	//Make sure string is not empty before using up an array spot.
	IF (StrLenA(pstData:= ADR(sShortString)) > 0) THEN
		TempArray[ArraySize] := sShortString;
		ArraySize := ArraySize + 1;
	END_IF

	//Remove copied components from long string
	StrDeleteA(
		pby:= ADR(StringIn), 
		iLength:= (iSplitLocation + LEN(SPLIT_CHAR)), 
		iPosition:= 1
	);

	//Check to see if more parameters can fit in array. If not exit loop
	IF (ArraySize > GPL_JSON.MAX_LEVELS) THEN
		EXIT;
	END_IF 
END_WHILE

ArraySize:= ArraySize - 1;

FOR i:= 0 TO ArraySize-1 DO
//reverse the order of the array
	VarNameArray[i+1].Name:= TempArray[ArraySize-i];	
END_FOR

SPLIT_VARNAME:= ArraySize;

END_FUNCTION

// Functions/JSONVALUE_TO_STRING
(*
| Author: Tim Van Meppelen, Pro Electric Inc.
| timv@proelectric.com
| Date: May 4, 2021
| convert a JSON value to string
*)
FUNCTION JSONVALUE_TO_STRING : STRING
VAR_INPUT
	In_JSON:		POINTER TO JSONVAR;
END_VAR

CASE In_JSON^.ValueType OF
JSONVALUETYPE.json_null:
	JSONVALUE_TO_STRING:= 'null';
JSONVALUETYPE.json_boolean:
	IF In_JSON^.Boolean THEN
		JSONVALUE_TO_STRING:= 'true';
	ELSE
		JSONVALUE_TO_STRING:= 'false';
	END_IF
JSONVALUETYPE.json_number:
	JSONVALUE_TO_STRING:= REAL_TO_STRING_X(In_JSON^.Number);
JSONVALUETYPE.json_integer:
	JSONVALUE_TO_STRING:= DINT_TO_STRING(In_JSON^.Integer);
JSONVALUETYPE.json_uinteger:
	CASE IN_JSON^.Format OF
	JSONFORMAT.Hex:
		JSONVALUE_TO_STRING:= UDINT_TO_HEXSTR(In_JSON^.UInteger);
	//TO DO:  other formats
	ELSE
		JSONVALUE_TO_STRING:= UDINT_TO_STRING(In_JSON^.UInteger);		
	END_CASE
JSONVALUETYPE.json_string:
	JSONVALUE_TO_STRING:= In_JSON^.CharString;
END_CASE

END_FUNCTION

// Functions/REAL_TO_STRING_X
(*
| Author: Tim Van Meppelen, Pro Electric Inc.
| timv@proelectric.com
| Date: Nov 2, 2018
| Standard REAL_TO_STRING function will always add a decimal place even if the input is a whole number
| this function will drop the ".0" on the string output
*)
FUNCTION REAL_TO_STRING_X : STRING
VAR_INPUT
	In_REAL:		REAL;
END_VAR
VAR
	TempVar:		STRING;
END_VAR

TempVar:= REAL_TO_STRING(In_REAL);
IF (RIGHT(STR:= TempVar, SIZE:= 2) = '.0') THEN
	REAL_TO_STRING_X:= DELETE(STR:= TempVar, LEN:= 2, POS:= LEN(TempVar) - 1);
ELSE
	REAL_TO_STRING_X:= TempVar;
END_IF

END_FUNCTION

// Functions/UDINT_TO_HEXSTR
(*
| Description:
| This function converts a UDINT (Unsigned Double Integer) value
| to its corresponding hexadecimal string representation (uppercase).
| 
| Example inputs/outputs: 255 -> '0xFF', 419 -> '0x1A3', 305419896 -> '0x12345678', 0 -> '0x0'
| 
| Limitations:
| - The returned string contains only valid hexadecimal digits (0-9, A-F), with '0x' prefix.
| - The output is always in uppercase.
| 
| Author: Fabrizio Morlino
| Date: 20/05/2025
*)
FUNCTION UDINT_TO_HEXSTR : STRING
VAR_INPUT
	udIn	: UDINT;
END_VAR
VAR
    i       : INT;
    nibble  : BYTE;
    result  : STRING(12) := '0x';
    hexchar : ARRAY[0..15] OF STRING(1) := ['0', '1', '2', '3', '4', '5', '6', '7', '8', '9','A', 'B', 'C', 'D', 'E', 'F'];
	xNotSkip: BOOL := FALSE;
END_VAR

// The FOR loop iterates through each nibble (4 bits) of the DWORD,
// starting from the most significant (bits 28-31) to the least significant (bits 0-3).
// 4 BYTE => 8 NIBBLE
FOR i := 7 TO 0 BY -1 DO
	nibble := TO_BYTE(SHR(udIn, i * 4) AND 16#F);
	// To write only the necessary digits (without zero-padding on the left)
	xNotSkip := xNotSkip OR nibble > 0 OR i = 0; //<= 1;
	IF xNotSkip THEN
		result := CONCAT(result, hexchar[nibble]);
	END_IF
END_FOR

UDINT_TO_HEXSTR := result;

END_FUNCTION

// Functions/STRING_TO_JSONVALUE
(*
| Author: Tim Van Meppelen, Pro Electric Inc.
| timv@proelectric.com
| Date: May 4, 2021
| Convert a string to a JSON value
*)
FUNCTION STRING_TO_JSONVALUE
VAR_INPUT
	In_String:		STRING(GPL_JSON.MAX_VALUE_SIZE);
	Out_JSON:		POINTER TO JSONVAR;
END_VAR
VAR
	TempBool:		BOOL;
	TempReal:		REAL;
	TempInt:		DINT;
	TempUint:		UDINT;
	Format:			JSONFORMAT;
END_VAR

IF (Out_JSON^.ValueType = JSONVALUETYPE.json_null) THEN
//if the type is not explicitly configured, make a guess at the type
//NOTE: this is used in JSON_TO_STRUCT to determine variable type
	Out_JSON^.ValueType:= VALUETYPE_FROM_STRING(In_String:= In_String, Format=> Format);
	OUT_JSON^.Format:= Format;	//helper var
END_IF

CASE Out_JSON^.ValueType OF
JSONVALUETYPE.json_null:
	Out_JSON^.Null:= 'null';
JSONVALUETYPE.json_boolean:
	StrToUpperA(pString:= ADR(In_String));
	IF (In_String = 'TRUE') THEN
		TempBool:= TRUE;
	ELSE
		TempBool:= FALSE;
	END_IF
	Out_JSON^.Boolean:= TempBool;
JSONVALUETYPE.json_integer:
	TempInt:= STRING_TO_DINT(In_String);
	Out_JSON^.Integer:= TempInt;
JSONVALUETYPE.json_uinteger:
	IF ISHEX(ADR(In_String)) THEN
		TempUInt:= HEXSTR_TO_UDINT(In_String);
	ELSE
		TempUint:= STRING_TO_UDINT(In_String);
	END_IF
	Out_JSON^.UInteger:= TempUInt;
JSONVALUETYPE.json_number:
	TempReal:= STRING_TO_REAL(In_String);
	Out_JSON^.Number:= TempReal;
JSONVALUETYPE.json_string:
	Out_JSON^.CharString:= In_String;
END_CASE

END_FUNCTION

// Functions/VALUETYPE_FROM_STRING
(*
| Author: Tim Van Meppelen, Pro Electric Inc.
| timv@proelectric.com
| Date: May 4, 2021
| take a guess at what kind of value this is based on what the string looks like
*)
FUNCTION VALUETYPE_FROM_STRING : JSONVALUETYPE
VAR_INPUT
	In_String:		STRING(GPL_JSON.MAX_VALUE_SIZE);
END_VAR
VAR_OUTPUT
	Format:			JSONFORMAT;
END_VAR

IF ISINTEGER(ADR(In_String)) THEN
	VALUETYPE_FROM_STRING:= JSONVALUETYPE.json_integer;
ELSIF ISNUMBER(ADR(In_String)) THEN
	VALUETYPE_FROM_STRING:= JSONVALUETYPE.json_number;
//NOTE:  UInteger type disabled because it's not
//necessarily possible to check for signed/unsigned from a string, where 
//the value could change.  Therefore, json_uinteger type must be manually configured
//ELSIF ISUINTEGER(ADR(In_String)) THEN
//	VALUETYPE_FROM_STRING:= JSONVALUETYPE.json_uinteger;	
ELSIF ISHEX(ADR(In_String)) THEN
	VALUETYPE_FROM_STRING:= JSONVALUETYPE.json_uinteger;
	Format:= JSONFORMAT.Hex;
ELSIF ISBOOLEAN(ADR(In_String)) THEN
	VALUETYPE_FROM_STRING:= JSONVALUETYPE.json_boolean;
ELSIF ISNULL(ADR(In_String)) THEN
	VALUETYPE_FROM_STRING:= JSONVALUETYPE.json_null;
ELSE
	VALUETYPE_FROM_STRING:= JSONVALUETYPE.json_string;
END_IF

END_FUNCTION

// Functions/ISINTEGER
(*
| Author: Tim Van Meppelen, Pro Electric Inc.
| timv@proelectric.com
| Date: Mar 2, 2020
| check if a string contains an integer, allows for "-" at the beginning of the string, and no decimals
*)
FUNCTION ISINTEGER : BOOL
VAR_INPUT
	In:				POINTER TO ARRAY[1..255] OF ASCII;
END_VAR
VAR
	i:				UINT;
	founddecimal:	BOOL;
END_VAR

FOR i:= 1 TO 255 DO
	CASE In^[i] OF 	
	ASCII.NULL:
	//end of string
		EXIT;
	ASCII.MINUS:
	//only allow a "-" in the first position	
		IF (i=1) THEN
			ISINTEGER:= TRUE;
		ELSE
			ISINTEGER:= FALSE;
			EXIT;
		END_IF
	ASCII.DOT:
	//no decimal points allowed in integers
		ISINTEGER:= FALSE;
		EXIT;
	ASCII._0..ASCII._9:
		ISINTEGER:= TRUE;
	ELSE
	//all other characters are not part of numbers
		ISINTEGER:= FALSE;
		EXIT;
	END_CASE
END_FOR

END_FUNCTION

// Functions/ISNUMBER
(*
| Author: Tim Van Meppelen, Pro Electric Inc.
| timv@proelectric.com
| Date: Oct 2, 2018
| check if a string contains a valid number, allows for "-" at the beginning of the string, and one "." character
| update June 9, 2025: allow for scientific notation
*)
FUNCTION ISNUMBER : BOOL
VAR_INPUT
	In:				POINTER TO ARRAY[1..255] OF ASCII;
END_VAR
VAR
    i                   : UINT;
    foundDecimal        : BOOL := FALSE;       // true after first '.'
    foundExponent       : BOOL := FALSE;       // true after first 'e' or 'E'
    insideExponent      : BOOL := FALSE;       // parsing the exponent section
    expSignAllowed      : BOOL := FALSE;       // '+' or '-' allowed only once just after 'e'
    expDigitFound       : BOOL := FALSE;       // at least one digit required after e/E
END_VAR

// -----------------------------------------------------------------------------
// Scan the string until the terminating ASCII.NULL (0x00) or buffer end.
// -----------------------------------------------------------------------------
FOR i := 1 TO 255 DO
    CASE In^[i] OF
    ASCII.NULL :             // reached end of string
        // valid only if we are not still waiting for exponent digits
        ISNUMBER := NOT insideExponent OR expDigitFound;
        RETURN;

    // -------------------------------------------------------------------------
    // Optional leading sign (only '-' is used in literal syntax, '+' is legal
    // in expressions but not required for a constant; keep '-' behaviour).
    // Inside exponent one optional '+' or '-' may follow immediately after 'e'.
    // -------------------------------------------------------------------------
    ASCII.MINUS, ASCII.PLUS :
        IF (i = 1) AND (In^[i] = ASCII.MINUS) THEN
            // leading '-' of mantissa
            ISNUMBER := TRUE;

        ELSIF insideExponent AND expSignAllowed THEN
            // sign belonging to exponent
            expSignAllowed := FALSE;  // consume it
        ELSE
            ISNUMBER := FALSE;
            RETURN;
        END_IF;

    // -------------------------------------------------------------------------
    // Decimal point allowed exactly once and only before the exponent.
    // -------------------------------------------------------------------------
    ASCII.DOT :
        IF foundDecimal OR insideExponent THEN
            ISNUMBER := FALSE; RETURN;
        END_IF;
        foundDecimal := TRUE;

    // -------------------------------------------------------------------------
    // Exponent marker ('e' or 'E') allowed once and must follow at least
    // one digit of the mantissa.
    // -------------------------------------------------------------------------
    ASCII._e_, ASCII._E :
        IF foundExponent THEN
            ISNUMBER := FALSE; RETURN;    // second exponent → invalid
        END_IF;
        foundExponent  := TRUE;
        insideExponent := TRUE;
        expSignAllowed := TRUE;           // allow one optional sign next
        expDigitFound  := FALSE;          // reset digit flag for exponent

    // -------------------------------------------------------------------------
    // Digits are always allowed; in exponent they satisfy the “at least one
    // digit” rule.
    // -------------------------------------------------------------------------
    ASCII._0..ASCII._9 :
        IF insideExponent THEN
            expDigitFound := TRUE;
            expSignAllowed := FALSE;      // any further '+'/'-' now illegal
        END_IF;
        ISNUMBER := TRUE;

    // -------------------------------------------------------------------------
    ELSE        // any other character invalidates the literal
        ISNUMBER := FALSE;
        RETURN;
    END_CASE
END_FOR
// If the loop ends without meeting ASCII.NULL, treat as “not a number”
ISNUMBER := FALSE;

END_FUNCTION

// Functions/ISHEX
(*
| Description:
| This function checks whether the input string is a valid hexadecimal value.
| The string may optionally start with '0x' or '0X'.
| Only characters 0-9, A-F, and a-f are considered valid (after the optional prefix).
| 
| Example inputs: 'FF' -> TRUE, '0xFF' -> TRUE, '1A3' -> TRUE, '0x123G' -> FALSE, '' -> FALSE
| 
| Limitations:
| - The maximum allowed length of the hexadecimal string (excluding '0x') is 8 characters.
| - Returns FALSE if the string is empty or contains invalid characters.
| 
| Author: Fabrizio Morlino
| Date: 20/05/2025
*)
FUNCTION ISHEX : BOOL
VAR_INPUT
	In	: POINTER TO ARRAY[1..255] OF ASCII;
END_VAR
VAR
	i	: UINT;
END_VAR

FOR i:= 1 TO 256 DO
	CASE In^[i] OF
	ASCII.NULL:
	//end of string
		EXIT;
	ASCII._x_:
	//only allow a "x" in the second position	
		IF (i=2) THEN
			ISHEX:= TRUE;
		ELSE
			ISHEX:= FALSE;
			EXIT;
		END_IF		
	ASCII._a_..ASCII._f_:
		ISHEX:= TRUE;
	ASCII._A..ASCII._F:
		ISHEX:= TRUE;
	ASCII._0..ASCII._9:
		ISHEX:= TRUE;
	ELSE // all other characters are not part of numbers
		ISHEX:= FALSE;
		EXIT;		
	END_CASE
END_FOR

END_FUNCTION

// Functions/ISBOOLEAN
(*
| Author: Tim Van Meppelen, Pro Electric Inc.
| timv@proelectric.com
| Date: Oct 2, 2018
| check if a string would convert to a valid boolean variable
*)
FUNCTION ISBOOLEAN : BOOL
VAR_INPUT
	In:			POINTER TO STRING(5);
END_VAR
VAR
	TempVar:	STRING(5);
END_VAR

TempVar:= In^;
StrToUpperA(pString:= ADR(TempVar));

ISBOOLEAN:= (TempVar = 'TRUE') OR (TempVar = 'FALSE');

END_FUNCTION

// Functions/ISNULL
(*
| Author: Tim Van Meppelen, Pro Electric Inc.
| timv@proelectric.com
| Date: June 5, 2025
| check if a string reads null
*)
FUNCTION ISNULL : BOOL
VAR_INPUT
	In:			POINTER TO STRING(4);
END_VAR
VAR
	TempVar:	STRING(4);
END_VAR

TempVar:= In^;
StrToUpperA(pString:= ADR(TempVar));

ISNULL:= (TempVar = 'NULL');

END_FUNCTION

// Functions/HEXSTR_TO_UDINT
(*
| Description:
| This function converts a string representing a hexadecimal number
| into a UDINT (Unsigned Double Integer) value.
| The string may optionally start with '0x' or '0X'.
| 
| Example inputs: 'FF' -> 255, '0xFF' -> 255, '1A3' -> 419, '0x12345678' -> 305419896
| 
| Limitations:
| - The maximum length of the hexadecimal string (excluding '0x') is 8 characters,
|   since a UDINT is a 32-bit integer (2^32 - 1), which corresponds to FFFFFFFF in hexadecimal.
| 
| Author: Fabrizio Morlino
| Date: 20/05/2025
*)
FUNCTION HEXSTR_TO_UDINT : UDINT
VAR_INPUT
    sHex 		: STRING; // Hex string to convert 
END_VAR
VAR_OUTPUT
	xError		: BOOL;
END_VAR
VAR
    i        	: INT;          // Index for iteration
    c        	: BYTE;         // Current character
    digit    	: BYTE;         // Numeric value of the hexadecimal character
    result   	: UDINT := 0;   // Final result
    sHexLen  	: INT;          // Length of the string
    startIdx 	: INT := 0;     // Start index after the prefix
END_VAR

// Removes the '0x' or '0X' prefix if present
IF (LEFT(sHex, 2) = '0x') OR (LEFT(sHex, 2) = '0X') THEN
    startIdx := 2;
END_IF;

sHexLen := LEN(sHex);

// If the string is empty after the prefix
IF sHexLen - startIdx <= 0 THEN
	xError := TRUE;
	RETURN;
END_IF

// If the hexadecimal string is too large for a UDINT
IF sHexLen - startIdx > 8 THEN
	xError := TRUE;
	RETURN;
END_IF

// Iterate through each character of the string
FOR i := startIdx TO sHexLen - 1 DO
    c := sHex[i];
    // Convert the character to a numeric value
    IF (c >= ASCII._0) AND (c <= ASCII._9) THEN
        digit := TO_BYTE(c) - ASCII._0;
    ELSIF (c >= ASCII._A) AND (c <= ASCII._F) THEN
        digit := TO_BYTE(c) - ASCII._A + 10;
    ELSIF (c >= ASCII._a_) AND (c <= ASCII._f_) THEN
        digit := TO_BYTE(c) - ASCII._a_ + 10;
    ELSE
        // Invalid character
		xError := TRUE;
        RETURN;
    END_IF;

    // Accumulate the result
    result := result * 16 + TO_UDINT(digit);
END_FOR;

// Returns the converted value
HEXSTR_TO_UDINT := result;

END_FUNCTION

// Functions/DWORD_TO_HEXSTR
(*
| Description:
| This function converts a UDINT (Unsigned Double Integer) value
| to its corresponding hexadecimal string representation (uppercase).
| 
| Example inputs/outputs: 255 -> '0xFF', 419 -> '0x1A3', 305419896 -> '0x12345678', 0 -> '0x0'
| modified to always return 4 decimals for unicode characters
| Limitations:
| - The returned string contains only valid hexadecimal digits (0-9, A-F), with '0x' prefix.
| - The output is always in uppercase.
| 
| Author: Fabrizio Morlino
| Date: 20/05/2025
*)
FUNCTION DWORD_TO_HEXSTR : STRING
VAR_INPUT
	dWIn	: DWORD;
END_VAR
VAR
    i       : INT;
    nibble  : BYTE;
    result  : STRING(12) := '0x';
    hexchar : ARRAY[0..15] OF STRING(1) := ['0', '1', '2', '3', '4', '5', '6', '7', '8', '9','A', 'B', 'C', 'D', 'E', 'F'];
	xNotSkip: BOOL := FALSE;
END_VAR

// The FOR loop iterates through each nibble (4 bits) of the DWORD,
// starting from the most significant (bits 28-31) to the least significant (bits 0-3).
// 4 BYTE => 8 NIBBLE
FOR i := 7 TO 0 BY -1 DO
	nibble := TO_BYTE(SHR(dWIn, i * 4) AND 16#F);
	// To write only the necessary digits (without zero-padding on the left)
	xNotSkip := xNotSkip OR nibble > 0 OR i = 0; //<= 1;
	IF xNotSkip THEN
		result := CONCAT(result, hexchar[nibble]);
	END_IF
END_FOR

DWORD_TO_HEXSTR := result;

END_FUNCTION

// Functions/DWORD_TO_UNICODE
(*
| Description:
| This function converts a UDINT (Unsigned Double Integer) value
| to its corresponding hexadecimal string representation (uppercase).
| 
| Example inputs/outputs: 255 -> '\uFF', 419 -> '\u1A3', 305419896 -> '0x12345678', 0 -> '\u0'
| 
| Limitations:
| - The returned string contains only valid hexadecimal digits (0-9, A-F), with '\u' prefix.
| - The output is always in uppercase.
| 
| Author: Fabrizio Morlino
| Date: 20/05/2025
*)
FUNCTION DWORD_TO_UNICODE : STRING
VAR_INPUT
	dWIn	: DWORD;
END_VAR
VAR
    i       : INT;
    nibble  : BYTE;
    result  : STRING(12) := '\u';
    hexchar : ARRAY[0..15] OF STRING(1) := ['0', '1', '2', '3', '4', '5', '6', '7', '8', '9','A', 'B', 'C', 'D', 'E', 'F'];
	xNotSkip: BOOL := FALSE;
END_VAR

// Always produce exactly 4 hex digits (nibble indices 3 down TO 0)
FOR i := 3 TO 0 BY -1 DO
    nibble := TO_BYTE( SHR(dWIn, i * 4) AND 16#F );
    result := CONCAT(result, hexchar[nibble]);
END_FOR

DWORD_TO_UNICODE := result;

END_FUNCTION

// Examples/ExampleJSON_PRG
(*
| Author: Tim Van Meppelen, Pro Electric Inc.
| timv@proelectric.com
| Date: Nov 2, 2018
| example program demonstrating JSONVAR, STRUCT_TO_JSON, AND JSON_TO_STRUCT
| 
| This example will populate a structure with values and types.  On a rising edge of ComposeJSON.Execute, 
| ComposeJSON will create a JSON string.  When ComposeJSON.Done is set, ParseJSON.Execute is set, and 
| ParseJSON will then parse that string back into a different structure.
*)
PROGRAM ExampleJSON_PRG
VAR
	ExampleJSONObj:		EXAMPLEJSONSTRUCT;
	ComposeJSON:		STRUCT_TO_JSON;
	JSONString:			STRING(1000);

	NewJSONObj:			EXAMPLEJSONSTRUCT;	
	ParseJSON:			JSON_TO_STRUCT;
	JSONString2:		STRING(1000);
	
	CreateJSONInFB:		EXAMPLE_FB;
END_VAR

ExampleJSONObj.var1.Boolean:= TRUE;
ExampleJSONObj.var2.Number:= 34.8756;
ExampleJSONObj.var3.CharString:= 'teststring';
ExampleJSONObj.obj.var4.Number:= 22;
ExampleJSONObj.obj.var5.AsString:= 'FALSE';	//JSONVAR will guess at type, in this case, boolean
ExampleJSONObj.obj.var6.CharString:= 'qwer';
ExampleJSONObj.obj.var7[1].Number:= 123.234;
ExampleJSONObj.obj.var7[2].AsString:= '55.46';	//JSONVAR will guess at type, in this case, a number
ExampleJSONObj.obj.var7[3].Number:= 985;
ExampleJSONObj.arrayobj[1].Number:= 1;
ExampleJSONObj.arrayobj[2].Number:= 2;
ExampleJSONObj.arrayobj[3].Number:= 3;

//create a JSON string from example object
ComposeJSON(
	JSONString:= ADR(JSONString), 
	JSONStringSize:= SIZEOF(JSONString),
	JSONVars:= ADR(ExampleJSONObj),
	NumberOfVars:= SIZEOF(ExampleJSONObj) / SIZEOF(JSONVAR)
);

//fill another example object with values from the created JSON string
ParseJSON(
	JSONString:= ADR(JSONString2), 
	JSONStringSize:= SIZEOF(JSONString2),
	JSONVars:= ADR(NewJSONObj),
	NumberOfVars:= SIZEOF(NewJSONObj) / SIZEOF(JSONVAR)
);

CreateJSONInFB();

END_PROGRAM

// Examples/EXAMPLE_FB
(*
| Author: Tim Van Meppelen, Pro Electric Inc.
| timv@proelectric.com
| Date: Jan 31, 2020
| example of use in a function block
*)
FUNCTION_BLOCK EXAMPLE_FB
VAR_INPUT
	MaxLevel:			INT;
END_VAR
VAR_OUTPUT
	Out:				STRING(255);
END_VAR
VAR
	color_temp:			JSONVAR;
	FirstScan:			BOOL:= TRUE;
	ComposeJSON:		STRUCT_TO_JSON;
END_VAR

color_temp.CharString:= 'red';

ComposeJSON(
	JSONString:= ADR(Out), 
	JSONStringSize:= SIZEOF(Out),
	JSONVars:= ADR(color_temp),
	NumberOfVars:= SIZEOF(color_temp) / SIZEOF(JSONVAR),
	MaxLevel:= MaxLevel
);

IF FirstScan THEN
	FirstScan:= FALSE;
	ComposeJSON.Execute:= TRUE;
END_IF

END_FUNCTION_BLOCK

// Functions/CLEANSTRING
(*
| Author: Tim Van Meppelen, Pro Electric Inc.
| timv@proelectric.com
| Date: Oct 9, 2018
| strip all control characters and spaces from a string
*)
FUNCTION CLEANSTRING : BOOL
VAR_INPUT
	StringPtr:		POINTER TO ARRAY[1..GPL_JSON.MAX_JSON_STRING] OF ASCII;
END_VAR
VAR
	i:				UINT;
	j:				UINT;
END_VAR

FOR i:= 1 TO GPL_JSON.MAX_JSON_STRING DO
	IF (StringPtr^[i] >= 1) AND (StringPtr^[i] <= 16#20) THEN
	//match all control and white space characters, except for null, which terminates a string
		FOR j:= i TO GPL_JSON.MAX_JSON_STRING DO
			IF (StringPtr^[j] = ASCII.NULL) THEN
			//null character terminates string
				EXIT;
			ELSE
			//shift character array left one
				StringPtr^[j]:= StringPtr^[j+1];
			END_IF
		END_FOR
		i:= i - 1;	//run loop at same position again
	ELSIF (StringPtr^[i] = ASCII.NULL) THEN
	//found null character at the end of the string
		EXIT;
	END_IF
END_FOR

CLEANSTRING:= TRUE;

END_FUNCTION

// Examples/Test_ArrayOfStruct_PRG
PROGRAM Test_ArrayOfStruct_PRG
VAR
	FirstScan:			BOOL:= TRUE;	
	
	LocalJSONObj:		ARRAYOFSTRUCT;
	ComposeJSON:		STRUCT_TO_JSON;
	JSONString:			STRING(255);

END_VAR

IF FirstScan THEN
	FirstScan:= FALSE;
	ComposeJSON.Execute:= TRUE;
END_IF

//create a JSON string
LocalJSONObj.arr[1].obj1.Number:= 23.5;
LocalJSONObj.arr[1]._obj2.Integer:= 3;
LocalJSONObj.arr[1].obj3.Boolean:= TRUE;

LocalJSONObj.arr[2].obj1.Number:= 54.5;
LocalJSONObj.arr[2]._obj2.Number:= 7.5;
LocalJSONObj.arr[2].obj3.Boolean:= FALSE;

LocalJSONObj.arr[3].obj1.Number:= 87.1;
LocalJSONObj.arr[3]._obj2.Integer:= 88;
LocalJSONObj.arr[3].obj3.Boolean:= TRUE;

LocalJSONObj.arr[4].obj1.Boolean:= FALSE;
LocalJSONObj.arr[4]._obj2.Number:= 132.55;
LocalJSONObj.arr[4].obj3.Integer:= 3;


ComposeJSON(
	JSONString:= ADR(JSONString), 
	JSONStringSize:= SIZEOF(JSONString),
	JSONVars:= ADR(LocalJSONObj),
	NumberOfVars:= SIZEOF(LocalJSONObj) / SIZEOF(JSONVAR)
);

END_PROGRAM

// Examples/Test_Array_PRG
PROGRAM Test_Array_PRG
VAR
	FirstScan:			BOOL:= TRUE;	
	
	testarray:			ARRAY[1..20] OF JSONVAR;
	ComposeJSON:		STRUCT_TO_JSON;
	JSONString:			STRING(255);
	
	NewString:			STRING(255):= '{"new":["234","34.5","98.4","10.4","812","5","23","65","95.6","98","234","34.5","98.4","10.4","812","5","23","65","95.6","98"]}';
	ParseJSON:			JSON_TO_STRUCT;
	new:				ARRAY[1..20] OF JSONVAR;	
END_VAR

IF FirstScan THEN
	FirstScan:= FALSE;
	ComposeJSON.Execute:= TRUE;
	ParseJSON.Execute:= TRUE;
END_IF

//create a JSON string
testarray[1].Number:= 32.5;
testarray[2].Number:= 65.2;
testarray[3].Number:= 81.54;
testarray[4].Number:= 1953.523;
testarray[5].Number:= 901.5;

ComposeJSON(
	JSONString:= ADR(JSONString), 
	JSONStringSize:= SIZEOF(JSONString),
	JSONVars:= ADR(testarray),
	NumberOfVars:= SIZEOF(testarray) / SIZEOF(JSONVAR)
);




//parse a JSON string and put it into a variable
ParseJSON(
	JSONString:= ADR(NewString), 
	JSONStringSize:= SIZEOF(NewString),
	JSONVars:= ADR(new),
	NumberOfVars:= SIZEOF(new) / SIZEOF(JSONVAR)
);

END_PROGRAM

// Examples/Test_NestedStruct_PRG
PROGRAM Test_NestedStruct_PRG
VAR
	FirstScan:			BOOL:= TRUE;	
	
	LocalJSONObj:		JSONSTRUCT_1;
	ComposeJSON:		STRUCT_TO_JSON;
	JSONString:			STRING(255);
	
	NewString:			STRING(255):= '{"new":{"obj1":"234", "obj2":"34.5", "obj3":"true","nest":{"obj1":"468.5", "obj2":"197", "obj3":"this is a string"}}}';
	ParseJSON:			JSON_TO_STRUCT;
	new:				JSONSTRUCT_1;
END_VAR

IF FirstScan THEN
	FirstScan:= FALSE;
	ComposeJSON.Execute:= TRUE;
	ParseJSON.Execute:= TRUE;
END_IF

//create a JSON string
LocalJSONObj.obj1.Number:= 23.5;
LocalJSONObj.obj2.Integer:= 3;
LocalJSONObj.obj3.Boolean:= TRUE;

ComposeJSON(
	JSONString:= ADR(JSONString), 
	JSONStringSize:= SIZEOF(JSONString),
	JSONVars:= ADR(LocalJSONObj),
	NumberOfVars:= SIZEOF(LocalJSONObj) / SIZEOF(JSONVAR)
);





//parse a JSON string and put it into a variable
ParseJSON(
	JSONString:= ADR(NewString), 
	JSONStringSize:= SIZEOF(NewString),
	JSONVars:= ADR(new),
	NumberOfVars:= SIZEOF(new) / SIZEOF(JSONVAR)
);

END_PROGRAM

// Examples/Test_SingleVar_PRG
PROGRAM Test_SingleVar_PRG
VAR
	FirstScan:			BOOL:= TRUE;	
	
	colour:				JSONVAR;	
	ComposeJSON:		STRUCT_TO_JSON;
	JSONString:			STRING(255);
	
	NewString:			STRING:= '{"color":"blue"}';
	ParseJSON:			JSON_TO_STRUCT;
	color:				JSONVAR;
END_VAR

IF FirstScan THEN
	FirstScan:= FALSE;
	ComposeJSON.Execute:= TRUE;
	ParseJSON.Execute:= TRUE;
END_IF

//create a JSON string from a variable
colour.CharString:= 'blue';
ComposeJSON(
	JSONString:= ADR(JSONString), 
	JSONStringSize:= SIZEOF(JSONString),
	JSONVars:= ADR(colour),
	NumberOfVars:= SIZEOF(colour) / SIZEOF(JSONVAR)
);



//parse a JSON string and put it into a variable
ParseJSON(
	JSONString:= ADR(NewString), 
	JSONStringSize:= SIZEOF(NewString),
	JSONVars:= ADR(color),
	NumberOfVars:= SIZEOF(color) / SIZEOF(JSONVAR)
);

END_PROGRAM

// Examples/Test_Struct_PRG
PROGRAM Test_Struct_PRG
VAR
	FirstScan:			BOOL:= TRUE;	
	
	LocalJSONObj:		JSONSTRUCT;
	ComposeJSON:		STRUCT_TO_JSON;
	JSONString:			STRING(255);
	
	NewString:			STRING:= '{"new":{"obj1":"234", "_obj2":"34.5", "obj3":"true"}}';
	ParseJSON:			JSON_TO_STRUCT;
	new:				JSONSTRUCT;
END_VAR

IF FirstScan THEN
	FirstScan:= FALSE;
	ComposeJSON.Execute:= TRUE;
	ParseJSON.Execute:= TRUE;
END_IF

//create a JSON string
LocalJSONObj.obj1.Number:= 23.5;
LocalJSONObj._obj2.Integer:= 3;
LocalJSONObj.obj3.Boolean:= TRUE;

ComposeJSON(
	JSONString:= ADR(JSONString), 
	JSONStringSize:= SIZEOF(JSONString),
	JSONVars:= ADR(LocalJSONObj),
	NumberOfVars:= SIZEOF(LocalJSONObj) / SIZEOF(JSONVAR)
);



//parse a JSON string and put it into a variable
ParseJSON(
	JSONString:= ADR(NewString), 
	JSONStringSize:= SIZEOF(NewString),
	JSONVars:= ADR(new),
	NumberOfVars:= SIZEOF(new) / SIZEOF(JSONVAR)
);

END_PROGRAM

// Functions/HEX4_TO_UINT
(*
| Author: Tim Van Meppelen, Pro Electric Inc.
| timv@proelectric.com
| Date: June 5, 2025
| convert 4 consecutive ASCII hex digits into a UINT
*)
FUNCTION HEX4_TO_UINT : UINT
VAR_INPUT
	{attribute 'displaymode':='hex'}
    pSrc 			: POINTER TO ARRAY[1..4] OF BYTE;	//first ASCII hex digit
END_VAR
VAR
    i        		: INT;
    nibble   		: UINT;
    result16 		: UINT := 0;
    ch       		: BYTE;
END_VAR

FOR i := 0 TO 3 DO
    ch := pSrc^[i];               (* read next digit                    *)
    CASE ch OF
	16#30..16#39 : // '0'–'9'
		nibble := TO_UINT(ch - 16#30);          
	16#41..16#46 : // 'A'–'F' 
		nibble := TO_UINT(ch - 16#37);          
	16#61..16#66 : //'a'–'f'
		nibble := TO_UINT(ch - 16#57);          
	ELSE  //not hex → treat as 0; caller can add range check
		nibble := 0;  
    END_CASE;
    result16 := SHL(result16, 4) OR nibble;
END_FOR
HEX4_TO_UINT := result16;

END_FUNCTION

// Functions/UINT_TO_HEX4
(*
| Author: Tim Van Meppelen, Pro Electric Inc.
| timv@proelectric.com
| Date: June 5, 2025
| Convert low 16 bits of code-point to 4 ASCII hex digits.  
| Caller ensures pDest→ARRAY[1..4] OF BYTE.
*)
FUNCTION UINT_TO_HEX4 : INT	//returns number of bytes written (1-3)
VAR_INPUT
    codePoint 	: UINT;
    pDest     	: POINTER TO ARRAY[1..4] OF BYTE;
END_VAR
VAR
    i      		: INT;
    nibble 		: UDINT;
END_VAR

FOR i := 0 TO 3 DO (* write high nibble first *)
    nibble := SHR(codePoint,((3 - i) * 4)) AND 16#F;
    IF nibble < 10 THEN
        pDest^[i + 1] := TO_BYTE(16#30 + nibble);   (* '0'–'9' *)
    ELSE
        pDest^[i + 1] := TO_BYTE(16#41 + (nibble - 10)); (* 'A'–'F' *)
    END_IF
END_FOR

UINT_TO_HEX4 := 4;

END_FUNCTION

// Visualizations/JSON_TO_STRUCT_VISU
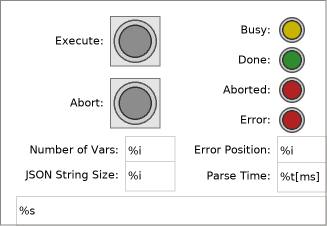
VISUALIZATION JSON_TO_STRUCT_VISU  // 327x226
(*
| Author: Tim Van Meppelen, Pro Electric Inc.
| timv@proelectric.com
| Date: Oct 31, 2023
| visualization for JSON_TO_STRUCT function block
| mostly used for testing
*)
VAR_IN_OUT
	ParseJSON:			JSON_TO_STRUCT;
END_VAR
    Lamp1 (277,15 30x30), variable: ParseJSON.Busy, style: Lamp-Lamp1-Yellow
    Label (177,15 100x30), "Busy:"
    Lamp1 (277,45 30x30), variable: ParseJSON.Done, style: Lamp-Lamp1-Green
    Label (177,45 100x30), "Done:"
    Lamp1 (277,75 30x30), variable: ParseJSON.Aborted, style: Lamp-Lamp1-Red
    Label (177,75 100x30), "Aborted:"
    Lamp1 (277,105 30x30), variable: ParseJSON.Error, style: Lamp-Lamp1-Red
    Label (177,105 100x30), "Error:"
    Label (177,135 100x30), "Error Position:"
    Textfield (277,136 50x30), "%i", text variable: ParseJSON.ErrorPosition
    Label (177,161 100x30), "Parse Time:"
    Textfield (277,162 50x30), "%t[ms]", text variable: ParseJSON.ParseTime
    Label (10,16 100x50), "Execute:"
    Label (10,78 100x50), "Abort:"
    PushSwitch (110,16 50x50), variable: ParseJSON.Execute, behaviour: TAP, style: Switch-PushSwitch-Gray
    PushSwitch (110,78 50x50), variable: ParseJSON.Abort, behaviour: TAP, style: Switch-PushSwitch-Gray
    Label (16,135 109x30), "Number of Vars:"
    Textfield (125,136 50x30), "%i", text variable: ParseJSON.NumberOfVars
    Textfield (125,161 50x30), "%i", text variable: ParseJSON.JSONStringSize
    Label (16,160 109x30), "JSON String Size:"
    Textfield (16,196 311x30), "%s", text variable: ParseJSON.ErrorMsg
END_VISUALIZATION

// Visualizations/STRUCT_TO_JSON_VISU
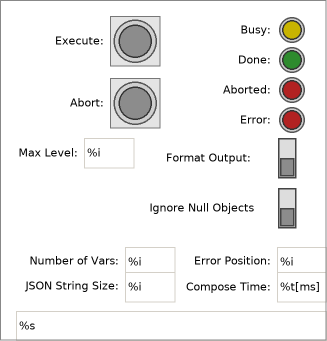
VISUALIZATION STRUCT_TO_JSON_VISU  // 327x341
(*
| Author: Tim Van Meppelen, Pro Electric Inc.
| timv@proelectric.com
| Date: Oct 31, 2023
| visualization for STRUCT_TO_JSON function block
| mostly used for testing
*)
VAR_IN_OUT
	ComposeJSON:			STRUCT_TO_JSON;
END_VAR
    Lamp1 (277,15 30x30), variable: ComposeJSON.Busy, style: Lamp-Lamp1-Yellow
    Label (177,15 100x30), "Busy:"
    Lamp1 (277,45 30x30), variable: ComposeJSON.Done, style: Lamp-Lamp1-Green
    Label (177,45 100x30), "Done:"
    Lamp1 (277,75 30x30), variable: ComposeJSON.Aborted, style: Lamp-Lamp1-Red
    Label (177,75 100x30), "Aborted:"
    Lamp1 (277,105 30x30), variable: ComposeJSON.Error, style: Lamp-Lamp1-Red
    Label (177,105 100x30), "Error:"
    Label (177,246 100x30), "Error Position:"
    Textfield (277,247 50x30), "%i", text variable: ComposeJSON.ErrorPosition
    Label (177,272 100x30), "Compose Time:"
    Textfield (277,272 50x30), "%t[ms]", text variable: ComposeJSON.ComposeTime
    Label (10,16 100x50), "Execute:"
    Label (10,78 100x50), "Abort:"
    PushSwitch (110,16 50x50), variable: ComposeJSON.Execute, behaviour: TAP, style: Switch-PushSwitch-Gray
    PushSwitch (110,78 50x50), variable: ComposeJSON.Abort, behaviour: TAP, style: Switch-PushSwitch-Gray
    Label (16,246 109x30), "Number of Vars:"
    Textfield (125,247 50x30), "%i", text variable: ComposeJSON.NumberOfVars
    Textfield (125,272 50x30), "%i", text variable: ComposeJSON.JSONStringSize
    Label (16,271 109x30), "JSON String Size:"
    Textfield (84,138 50x30), "%i", text variable: ComposeJSON.MaxLevel
        OnMouseClick: write the text variable via Default
    Label (10,138 74x30), "Max Level:"
    Label (157,138 100x40), "Format Output:"
    Textfield (16,311 311x30), "%s", text variable: ComposeJSON.ErrorMsg
    DipSwitch (267,138 40x40), variable: ComposeJSON.Format, behaviour: TOGGLE, style: Switch-DipSwitch-Gray
    DipSwitch (267,188 40x40), variable: ComposeJSON.IgnoreNull, behaviour: TOGGLE, style: Switch-DipSwitch-Gray
    Label (99,188 158x40), "Ignore Null Objects"
END_VISUALIZATION

// Visualizations/JSONVARS_TABLE_VISU
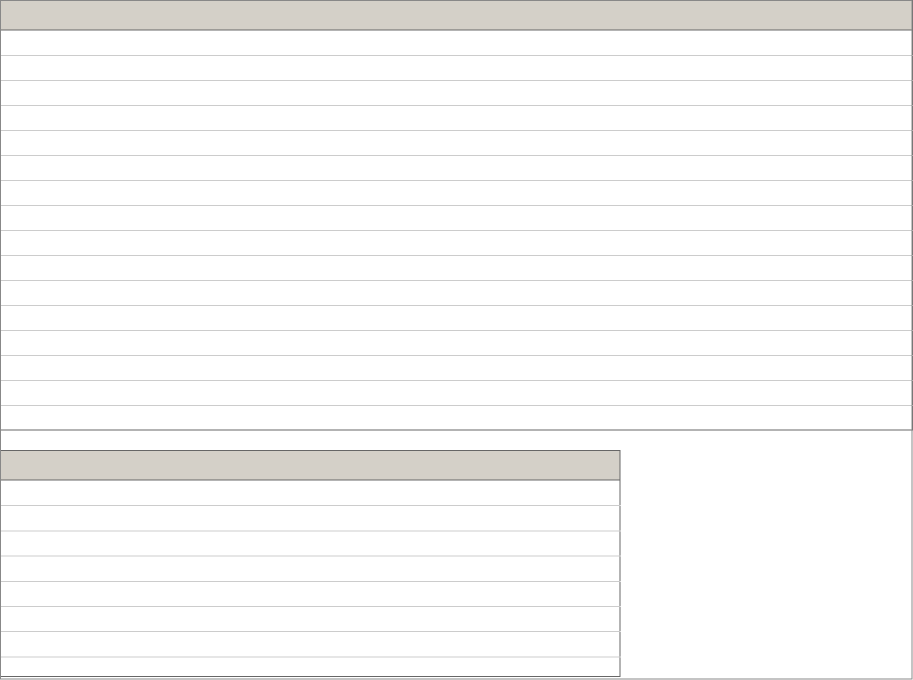
VISUALIZATION JSONVARS_TABLE_VISU  // 913x680
(*
| Author: Tim Van Meppelen, Pro Electric Inc.
| timv@proelectric.com
| Date: Dec 6, 2023
| Visu to show the attributes of JSONVARS, for testing and troubleshooting
| NOTE:  this visu will not work in simulation mode, at least in ESME 2.1.1, I haven't tested any other environmens
*)
VAR_IN_OUT
	JSONVars:			POINTER TO ARRAY[1..GPL_JSON.MAX_VARS] OF JSONVAR;	//pointer to local structure made up of type JSONVAR
	NumberOfVars:		UDINT;		//number of variables in the local structure or array
END_VAR
VAR
	SelectedVar:		INT:= 1;
END_VAR
    Table (0,0 913x430), data array: JSONVars
        p1128707560: NumberOfVars
        p1014161805: GPL_JSON.MAX_VARS - 1 + 1
        p1137915858: SelectedVar
        p3854506369: JSONVars^[INDEX].Names
        p1892666644: JSONVars^[INDEX]._VarNameFull
        p338671338: JSONVars^[INDEX]._ValueType
        p2170511999: JSONVars^[INDEX]._InternalValue
        p3723444502: JSONVars^[INDEX]._Size
        p1218418051: JSONVars^[INDEX]._ApplicationLevel
        p746581629: JSONVars^[INDEX]._InitDone
        p3104783080: JSONVars^[INDEX]._LastIndex
        p2501879983: JSONVars^[INDEX].HMIVarAsString
        p7306298: JSONVars^[INDEX].PrevApplicationLevel
        p1933151965: JSONVars^[INDEX].PrevNameArray
        p3863566920: JSONVars^[INDEX].VarName
        p2192122294: JSONVars^[INDEX].ProgramLevel
        p400160035: JSONVars^[INDEX].AsString
        p3726181087: JSONVars^[INDEX].CharString
        p3136911649: JSONVars^[INDEX].Init
        p797552052: JSONVars^[INDEX].Integer
        p60375027: JSONVars^[INDEX].LastIndex
        p2531912550: JSONVars^[INDEX].Null
        p693678525: JSONVars^[INDEX].Number
        p3156763944: JSONVars^[INDEX].Size
        p511219082: Var Name
        p2319025000: Prg Level
        p290089404: JSONVars^[INDEX].AsDateTime
        p4236254150: JSONVars^[INDEX].Boolean
        p3286028342: JSONVars^[INDEX].ApplicationLevel
        p3718605203: JSONVars^[INDEX].ValueType
    Frame (0,450 620x230)
        shows JSONVAR_TABLE_VISU(JSON_Var := JSONVars^[SelectedVar])
END_VISUALIZATION

// Visualizations/JSONVAR_TABLE_VISU
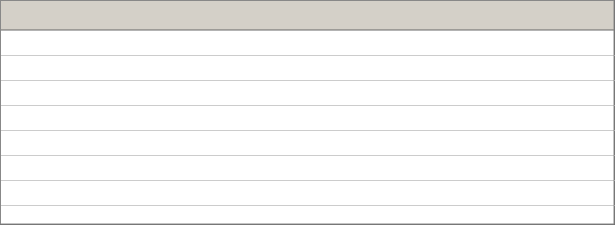
VISUALIZATION JSONVAR_TABLE_VISU  // 615x225
VAR_IN_OUT
	JSON_Var:		JSONVAR;
END_VAR
    Table (0,0 615x225), data array: JSON_Var.JSONVarInfo
        p3104783080: JSON_Var.JSONVarInfo[INDEX].EndArray
        p2501879983: JSON_Var.HMIVarAsString
        p7306298: JSON_Var.PrevApplicationLevel
        p1933151965: JSON_Var.PrevNameArray
        p3863566920: JSON_Var.ApplicationLevel
        p2192122294: JSON_Var.AsDateTime
        p400160035: JSON_Var.AsString
        p1265227338: JSON_Var.Boolean
        p3726181087: JSON_Var.CharString
        p3136911649: JSON_Var.Init
        p797552052: JSON_Var.Integer
        p60375027: JSON_Var.LastIndex
        p2531912550: JSON_Var.Null
        p693678525: JSON_Var.Number
        p3156763944: JSON_Var.Size
        p3636993750: JSON_Var.ValueType
        p1303956035: JSON_Var.VarName
        p4088588272: End Arr
        p1014161805: GPL_JSON.MAX_LEVELS - 1 + INT#1
        p3854506369: JSON_Var.JSONVarInfo[INDEX].Name
        p1892666644: JSON_Var.JSONVarInfo[INDEX].NewObject
        p338671338: JSON_Var.JSONVarInfo[INDEX].InObject
        p2170511999: JSON_Var.JSONVarInfo[INDEX].EndObject
        p1218418051: JSON_Var.JSONVarInfo[INDEX].NewArray
        p746581629: JSON_Var.JSONVarInfo[INDEX].InArray
        p511219082: New Obj
        p1755163831: In Obj
        p4092479075: End Obj
        p505689113: New Arr
        p1757482276: In Arr
        p4008173056: JSON_Var.JSONVarInfo[INDEX].ArrayIndex
END_VISUALIZATION

(* text list ValueType_Textlist (id | default)
  0 | string
  1 | number
  2 | integer
  3 | unsigned int
  4 | hex
  5 | boolean
  6 | null
  7 | array
  8 | object
   |  *)
